(*********************************** G.D S.p.A. - Technical Department ***********************************
============= PROGRAM INFO ============
FOLDER:             TBD
MACHINES INVOLVED:  TBD 

============= DESCRIPTION =============
csp machine declaration

============= REVISIONS ===============
Date		Version	 	Author      	Description             
----------	-------		------------  	--------------------------------------------
2019/04/05 	0000.00	 	M.Grasso		Creation of the PRG

**********************************************************************************************************)
(*$R process_ref := prc; $*)
PROGRAM csp_case_loader_guide
VAR
	
	prc:											process;
	prc_path:										STRING;
	
END_VAR

_read_var_input();

_object_manager();

IF NOT objects_running()
THEN
	RETURN;	
END_IF

_read_process_image();

_mode_manager();

_set_runtime_properties();

(********************************* BODY *********************************)
(************************************************************************)

_handle_messages();

_write_output();

ACTION _handle_messages:
;
END_ACTION

ACTION _handle_process_test:
;
END_ACTION

ACTION _mode_manager:
IF process_mode_req_is_pending(prc)
THEN
    process_apply_mode_req_first_step(prc);
    CASE process_get_mode(prc) OF
        MODE_TO_ABSENT:
			;
        MODE_TO_INACTIVE:
			;
        MODE_TO_TEST:
			;
        MODE_TO_OPERATIONAL:
			;
    END_CASE
    process_apply_mode_req_second_step(prc);
END_IF
END_ACTION

ACTION _object_manager:
IF objects_initialization()
THEN
	sub_process_init(
		object_name					:= 'csp_case_loader_guide.prc', 
		process						:= csp_case_loader.prc, 
		CONVERSION_this				:= prc);
		
	prc_path 						:= process_get_path(prc);
END_IF

IF objects_running()
THEN
	process_cycle(prc);
END_IF
END_ACTION

ACTION _read_process_image:
;
END_ACTION

ACTION _read_var_input:
;
END_ACTION

ACTION _set_runtime_properties:
;
END_ACTION

ACTION _write_output:
;
END_ACTION

END_PROGRAM

(* stored: Version 1.1.0.1, ProductVersion 3.1.4022.12
   POU csp_case_loader_guide: Id {dc1118d7-97b8-4996-b79d-526eaf90a474}, SpecialFunc None
   Action _handle_messages: Id {5889af7c-56f9-4f93-a56c-088d08f75988}
   Action _handle_process_test: Id {140636af-5361-4a75-8a36-fc99680f071d}
   Action _mode_manager: Id {c8ea7a23-dc87-4a40-9a87-92ab0e27c123}
   Action _object_manager: Id {c7643ce7-6c83-45f9-939c-8b7d2418cab4}
   Action _read_process_image: Id {72b9a15a-85fe-419b-ab38-3ff365531ae4}
   Action _read_var_input: Id {b56b081e-19bb-4a5f-96bd-d3448c9b9d92}
   Action _set_runtime_properties: Id {733c135d-9797-482b-a52e-5a371bc73cbd}
   Action _write_output: Id {18024588-2198-444d-acdd-33898eba190e} *)
